TYPE stMachineParams :
STRUCT
	iErrorPimOffset			: INT;
	bPartsCount				: BOOL := TRUE;
END_STRUCT
END_TYPE

(* stored: Version 1.1.0.1, ProductVersion 3.1.4024.13
   DUT stMachineParams: Id {bbd270ac-8f33-41e1-8a4b-740bd07cf388} *)
